# EPICS autosave request: GalilSup/Db/galil_dmc_ctrl.req
# Controller settings
$(P)LIMITTYPE_CMD.VAL
$(P)HOMETYPE_CMD.VAL
$(P)HOMEEDGE_CMD.VAL
$(P)DEFER_MODE_CMD.VAL
$(P)ECATNETWORK_CMD
